// TIA Portal V20 export
TYPE "UDT_Service_ProzessValueMapping"
   STRUCT
      Mapping { ExternalAccessible := 'False'; ExternalVisible := 'False'; ExternalWritable := 'False'} : Int := -1;
   END_STRUCT;
END_TYPE
